FUNCTION_BLOCK FB_Trennen EXTENDS FB_Basis
VAR_INPUT
	Reaktor			:I_Reaktor;
	Auswertung		:I_Auswertung;
END_VAR
VAR_OUTPUT
END_VAR
VAR
	
END_VAR

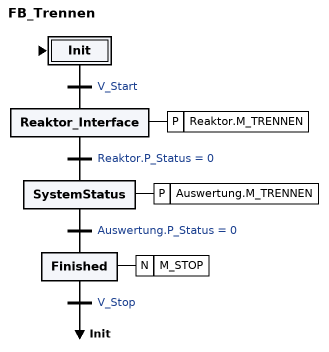
INITIAL_STEP Init:
END_STEP
TRANSITION FROM Init TO Reaktor_Interface
    := V_Start;
END_TRANSITION
STEP Reaktor_Interface:
    Reaktor.M_TRENNEN(P);
END_STEP
TRANSITION FROM Reaktor_Interface TO SystemStatus_
    := Reaktor.P_Status = 0;
END_TRANSITION
STEP SystemStatus_:  // name as stored: SystemStatus 
    Auswertung.M_TRENNEN(P);
END_STEP
TRANSITION FROM SystemStatus_ TO Finished
    := Auswertung.P_Status = 0;
END_TRANSITION
STEP Finished:
    M_STOP(N);
END_STEP
TRANSITION FROM Finished TO Init
    := V_Stop;
END_TRANSITION

END_FUNCTION_BLOCK

(* stored: Version 1.1.0.1, ProductVersion 3.1.4024.12
   POU FB_Trennen: Id {0c18d517-b5da-44ce-9946-78fd1fdd29bf}, SpecialFunc None *)
